TYPE ST_LOG_RejectReasons :
STRUCT
	(*nRejectID			: INT;
 	sMETSRejectCode		: STRING(50);*)
	nRejectCounter		: UINT;
	stLastTimeStamp		: TIMESTRUCT;
END_STRUCT
END_TYPE

(* stored: Version 1.1.0.1
   DUT ST_LOG_RejectReasons: Id {54e7a6f9-bcf4-4f55-b55c-beb1c83fd015} *)
